
// ===== library types =====

TYPE "UDT_Node_Universal_G2"
   STRUCT
      Enable : Bool := FALSE;   // Enable polling for this slave node (TRUE = Active)
      SlaveAddress : UInt := 1;   // Modbus RTU slave address (1..247)
      SwapWords : Bool := FALSE;
      Requests : Array[1..10] of "UDT_Request_Universal_G2";   // Data Address Of Slave Device
   END_STRUCT;
END_TYPE

TYPE "UDT_Request_Universal_G2"
   STRUCT
      Enable : Bool := FALSE;   // Enable or disable this specific request (TRUE = Active)
      Mode : USInt := 1;   // Modbus function mode (0: Read, 1: Write)
      DataAddress : UDInt := 40001;   // Modbus register start address (e.g., 40001, 30001)
      DataLen : UInt := 1;   // Number of registers to read/write (Max 10 )
      IsDouble : Bool := FALSE;   // False = 16-bit, True = 32-bit
      DataValue : Array[0..9] of DWord;   // Data value to write to slave or value received from slave
      Done : Bool := FALSE;   // Execution status (TRUE = Request completed successfully)
      Error : Bool := FALSE;   // Execution status (TRUE = Request failed or timed out)
      Status : Word := 16#0;   // Modbus status code / error code from MB_MASTER
   END_STRUCT;
END_TYPE

TYPE "UDT_Convert"
   STRUCT
      DataValue_INT : Array[1..10] of Int;
      DataValue_DINT : Array[1..10] of DInt;
      DataValue_REAL : Array[1..10] of Real;
   END_STRUCT;
END_TYPE

FUNCTION_BLOCK "DataConverter"   // FB2, LAD
{ S7_Optimized_Access := 'TRUE' }
VERSION : 0.1
   VAR_INPUT
      Node_ID : USInt := 0;   // Target Modbus Node ID for processing
      Start_Req : Int := 0;   // Start index for request processing range
      End_Req : Int := 0;   // End index for request processing range
      Enable_Write : Bool := FALSE;
   END_VAR
   VAR_IN_OUT
      Nodes : Array[*] of "UDT_Node_Universal_G2";   // Slave Name
   END_VAR
   VAR
      Requests : Array[1..10] of "UDT_Convert";   // Data storage for HMI mapping using custom UDT
      Temp : Bool;
      req_idx : Int;   // Loop index for iterating through requests
      data_idx : Int;   // Loop index for iterating through data values
      current_mode : USInt;   // Temporary storage for current request mode (0=Read, 1=Write)
      current_len : UInt;   // Temporary storage for current data length
      is_double : Bool;   // Flag indicating if current data is 32-bit
      temp_dword : DWord;   // Temporary memory for 32-bit data casting
      offset : Int;   // Offset calculation for 32-bit Modbus registers
      min_idx : DInt;
      max_idx : DInt;
      swap_words : Bool;
   END_VAR
BEGIN

REGION Network 2 (SCL)
   // 1. استخراج محدوده آرایه دینامیک نودها از پین InOut
   #min_idx := LOWER_BOUND(ARR := #Nodes, DIM := 1);
   #max_idx := UPPER_BOUND(ARR := #Nodes, DIM := 1);

   // 2. بررسی اینکه Node_ID وارد شده در محدوده مجاز باشد
   IF USINT_TO_DINT(#Node_ID) >= #min_idx AND USINT_TO_DINT(#Node_ID) <= #max_idx THEN

       // 3. بررسی فعال بودن نود انتخاب شده
       IF #Nodes[#Node_ID].Enable THEN

           // 4. حلقه پیمایش درخواستها
           FOR #req_idx := LIMIT(MN := 1, IN := #Start_Req, MX := 10) TO LIMIT(MN := 1, IN := #End_Req, MX := 10) DO

               // 5. بررسی فعال بودن درخواست جاری
               IF #Nodes[#Node_ID].Requests[#req_idx].Enable THEN

                   // کش کردن پارامترهای درخواست برای سرعت بالا
                   #current_mode := #Nodes[#Node_ID].Requests[#req_idx].Mode;
                   #current_len := #Nodes[#Node_ID].Requests[#req_idx].DataLen;
                   #is_double := #Nodes[#Node_ID].Requests[#req_idx].IsDouble;

                   // محدودسازی طول دیتا (محافظت در برابر خطای طول آرایه)
                   IF #current_len > 10 THEN
                       #current_len := 10;
                   END_IF;

                   IF #current_len > 0 THEN

                       // 6. حلقه پردازش عناصر دیتا
                       FOR #data_idx := 0 TO UINT_TO_INT(#current_len) - 1 DO

                           #offset := #data_idx + 1;

                           // ==========================================
                           // Mode 0: READ (از Modbus به HMI)
                           // ==========================================
                           IF #current_mode = 0 THEN

                               #temp_dword := #Nodes[#Node_ID].Requests[#req_idx]."DataValue"[#data_idx];

                               // تبدیل و انتقال مستقیم دیتا 
                               IF NOT #is_double THEN
                                   #Requests[#req_idx].DataValue_INT[#offset] := DWORD_TO_INT(#temp_dword);
                               ELSE
                                   #Requests[#req_idx].DataValue_DINT[#offset] := DWORD_TO_DINT(#temp_dword);
                                   #Requests[#req_idx].DataValue_REAL[#offset] := DWORD_TO_REAL(#temp_dword);
                               END_IF;

                               // ==========================================
                               // Mode 1: WRITE (از HMI به Modbus)
                               // شرط اضافه شده: بررسی روشن بودن Enable_Write
                               // ==========================================
                           ELSIF (#current_mode = 1) AND #Enable_Write THEN

                               // تشخیص هوشمند نوع دیتا بر اساس مقدار غیر صفر
                               IF #Requests[#req_idx].DataValue_REAL[#offset] <> 0.0 THEN
                                   // اولویت اول: اگر مقدار REAL غیر صفر بود
                                   #temp_dword := REAL_TO_DWORD(#Requests[#req_idx].DataValue_REAL[#offset]);

                               ELSIF #Requests[#req_idx].DataValue_DINT[#offset] <> 0 THEN
                                   // اولویت دوم: اگر مقدار DINT غیر صفر بود
                                   #temp_dword := DINT_TO_DWORD(#Requests[#req_idx].DataValue_DINT[#offset]);

                               ELSIF #Requests[#req_idx].DataValue_INT[#offset] <> 0 THEN
                                   // اولویت سوم: اگر مقدار INT غیر صفر بود
                                   #temp_dword := INT_TO_DWORD(#Requests[#req_idx].DataValue_INT[#offset]);

                               ELSE
                                   // اگر همه صفر بودند
                                   #temp_dword := 16#0000_0000;
                               END_IF;

                               // انتقال دیتای نهایی به بافر ارسال مدباس
                               #Nodes[#Node_ID].Requests[#req_idx]."DataValue"[#data_idx] := #temp_dword;

                           END_IF;

                       END_FOR; // پایان حلقه دیتا
                   END_IF;

               END_IF;

           END_FOR; // پایان حلقه رکویستها

       END_IF;
   END_IF;
END_REGION
END_FUNCTION_BLOCK